(* Logix 5000 project; controller WWTP_SOLIDS_CLX vendor 1 type 14 code 54 rev 17.2; software revision 17.00; part 10 of 16 *)
(* tags used below, declared in another part *)
   Inp_PermOK : BOOL;   // 1=Permissives OK, motor can start
   Inp_NBPermOK : BOOL;   // 1=Non-Bypassable Permissives OK, motor can start
   Inp_IntlkOK : BOOL;   // 1=Interlocks OK, motor can start/run
   Inp_NBIntlkOK : BOOL;   // 1=Non-Bypassable Interlocks OK, motor can start/run
   Inp_IOFault : BOOL;   // Input Communication Status 0=OK, 1=fail
   Inp_Sim : BOOL;   // 1=Simulate working motor; 0=Start/Stop/ Monitor actual motor
   Cfg_UseRunFdbk : BOOL;   // 1=Motor run feedback should be used for failure checking
   Cfg_PCmdClear : BOOL;   // 1=Clear Program Commands on receipt 0=Leave Set
   Cfg_HasIntlkTripAlm : BOOL;   // 1=Interlock Trip Alarm exists and will be checked
   Cfg_HasIOFaultAlm : BOOL;   // 1=I/O Fault Alarm exists and will be checked
   PSet_Owner : DINT;   // Program Owner Request ID (non-zero) or Release (zero)
   PCmd_Start : BOOL;   // Program Command to Start Motor
   PCmd_Stop : BOOL;   // Program Command to Stop Motor
   PCmd_Acq : BOOL;   // Program Command to Acquire ownership (Oper/OOS to Prog)
   PCmd_Rel : BOOL;   // Program Command to Release ownership (Prog to OOS)
   PCmd_Lock : BOOL;   // Program Command to Lock Mode in Prog
   PCmd_Unlock : BOOL;   // Program Command to Unlock Mode
   PCmd_FailToStartInhibit : BOOL;   // Program Command to Inhibit Fail to Start Alarm
   PCmd_FailToStartUninhibit : BOOL;   // Program Command to Uninhibit Fail to Start Alarm
   PCmd_FailToStopInhibit : BOOL;   // Program Command to Inhibit Fail to Stop Alarm
   PCmd_FailToStopUninhibit : BOOL;   // Program Command to Uninhibit Fail to Stop Alarm
   PCmd_IntlkTripInhibit : BOOL;   // Program Command to Inhibit Interlock Trip Alarm
   PCmd_IntlkTripUninhibit : BOOL;   // Program Command to Uninhibit Interlock Trip Alarm
   PCmd_IOFaultInhibit : BOOL;   // Program Command to Inhibit I/O Fault Alarm
   PCmd_IOFaultUninhibit : BOOL;   // Program Command to Uninhibit I/O Fault Alarm
   OCmd_Start : BOOL;   // Operator Command to Start Motor
   OCmd_Stop : BOOL;   // Operator Command to Stop Motor
   OCmd_Bypass : BOOL;   // Operator Command to Bypass all Bypassable Interlocks and Permissives
   OCmd_Check : BOOL;   // Operator Command to Check (not bypass) all Interlocks and Permissives
   MCmd_Disable : BOOL;   // Maintenance Command to Disable Motor
   MCmd_Enable : BOOL;   // Maintenance Command to Enable (allow to run) Motor
   Val_Owner : DINT;   // Current Object Owner ID (0=not owned)
   Val_Notify : SINT;   // Current Alarm Level and Acknowledgement (enumeration)
   Sts_Stopped : BOOL;   // 1=Motor requested to stop and is confirmed stopped
   Sts_Starting : BOOL;   // 1=Motor requested to run and awaiting run feedback
   Sts_Running : BOOL;   // 1=Motor requested to run and is confirmed running
   Sts_Stopping : BOOL;   // 1=Motor requested to stop and awaiting stopped feedback
   Sts_Available : BOOL;   // 1=Motor available for control by automation (Prog)
   Sts_Bypass : BOOL;   // 1=Bypassable Interlocks and Permissives are Bypassed
   Sts_BypActive : BOOL;   // 1=Bypassing Active (Bypassed or Maintenance)
   Sts_Disabled : BOOL;   // 1=Motor is Disabled
   Sts_Hand : BOOL;   // 1=Mode is Hand (supersedes Maint, Ovrd, Prog, Oper)
   Sts_Maint : BOOL;   // 1=Mode is Maintenance (supersedes Ovrd, Prog, Oper)
   Sts_Prog : BOOL;   // 1=Mode is Program (auto)
   Sts_Oper : BOOL;   // 1=Mode is Operator (manual)
   Sts_FailToStop : BOOL;   // 1=Motor Failed to Stop
   Alm_IntlkTrip : BOOL;   // 1=Alarm: Motor stopped by an Interlock NOT OK
   Ack_IntlkTrip : BOOL;   // 1=Interlock Trip Alarm has been acknowledged
   Sts_IntlkTripDisabled : BOOL;   // 1=Interlock Trip Alarm is Disabled (not saved or sent)
   Sts_IntlkTripInhibited : BOOL;   // 1=Interlock Trip Alarm has been inhibited by logic
   Sts_IntlkTripSuppressed : BOOL;   // 1=Interlock Trip Alarm has been suppressed (logged only)
   Alm_IOFault : BOOL;   // 1=I/O Fault Alarm
   Ack_IOFault : BOOL;   // 1=I/O Fault Alarm has been acknowledged
   Sts_IOFaultDisabled : BOOL;   // 1=I/O Fault Alarm is Disabled (not saved or sent)
   Sts_IOFaultInhibited : BOOL;   // 1=I/O Fault Alarm has been inhibited by logic
   Sts_IOFaultSuppressed : BOOL;   // 1=I/O Fault Alarm has been suppressed (logged only)
   Rdy_Start : BOOL;   // 1=Ready to receive OCmd_Start (enables HMI button)
   Rdy_Stop : BOOL;   // 1=Ready to receive OCmd_Stop (enables HMI button)
   Rdy_Bypass : BOOL;   // 1=Ready to receive OCmd_Bypass (enables HMI button)
   Rdy_Check : BOOL;   // 1=Ready to receive OCmd_Check (enables HMI button)
   Rdy_Disable : BOOL;   // 1=Ready to receive MCmd_Disable (enables HMI button)
   Rdy_Enable : BOOL;   // 1=Ready to receive MCmd_Enable (enables HMI button)
   Mode : P_Mode;   // Motor Mode Selection
   IOFault : P_Alarm;   // I/O Fault Alarm
   IntlkTrip : P_Alarm;   // Interlock Trip Alarm
   FailToStop : P_Alarm;   // Motor Failed to Stop Alarm
   FailToStart : P_Alarm;   // Motor Failed to Start Alarm
   Wrk_Run : BOOL;   // 1=Motor should be "running", 0=should be "stopped"
   Wrk_Fault : BOOL;   // 1=a Motor Fault has been detected
   Wrk_RunFdbk : BOOL;   // Run Feedback based on mode, simulation, etc. 1=running
   Wrk_Notify : DINT;   // Buffer for building Val_Notify
   Wrk_Disabled : BOOL;   // Internal Motor is Disabled
(* P_Motor, continued *)

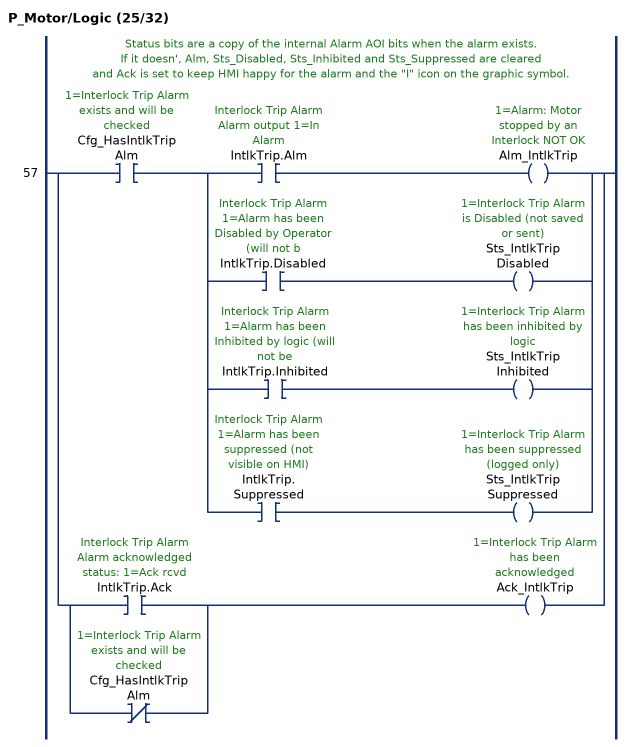
   // Status bits are a copy of the internal Alarm AOI bits when the alarm exists.
   // If it doesn', Alm, Sts_Disabled, Sts_Inhibited and Sts_Suppressed are cleared
   // and Ack is set to keep HMI happy for the alarm and the "I" icon on the graphic symbol.
   57: [XIC(Cfg_HasIntlkTripAlm) [XIC(IntlkTrip.Alm) OTE(Alm_IntlkTrip) ,XIC(IntlkTrip.Disabled) OTE(Sts_IntlkTripDisabled) ,XIC(IntlkTrip.Inhibited) OTE(Sts_IntlkTripInhibited) ,XIC(IntlkTrip.Suppressed) OTE(Sts_IntlkTripSuppressed) ] ,[XIC(IntlkTrip.Ack) ,XIO(Cfg_HasIntlkTripAlm) ] OTE(Ack_IntlkTrip) ];
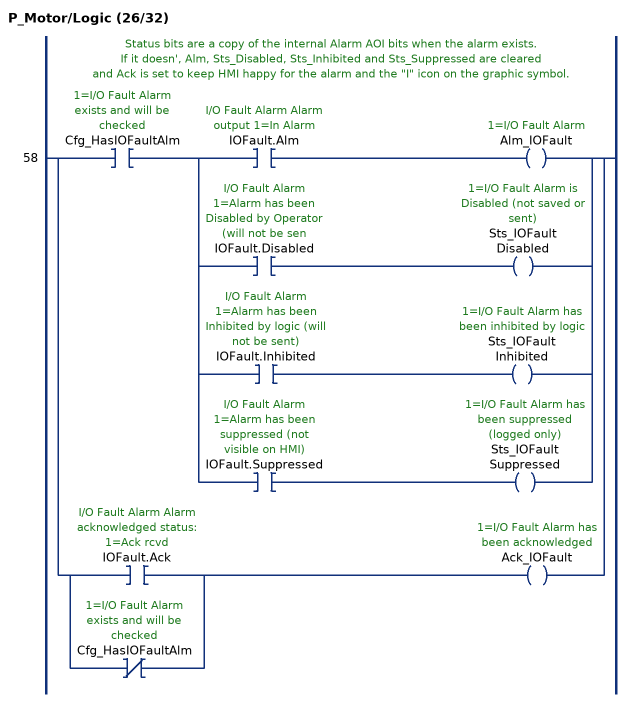
   // Status bits are a copy of the internal Alarm AOI bits when the alarm exists.
   // If it doesn', Alm, Sts_Disabled, Sts_Inhibited and Sts_Suppressed are cleared
   // and Ack is set to keep HMI happy for the alarm and the "I" icon on the graphic symbol.
   58: [XIC(Cfg_HasIOFaultAlm) [XIC(IOFault.Alm) OTE(Alm_IOFault) ,XIC(IOFault.Disabled) OTE(Sts_IOFaultDisabled) ,XIC(IOFault.Inhibited) OTE(Sts_IOFaultInhibited) ,XIC(IOFault.Suppressed) OTE(Sts_IOFaultSuppressed) ] ,[XIC(IOFault.Ack) ,XIO(Cfg_HasIOFaultAlm) ] OTE(Ack_IOFault) ];
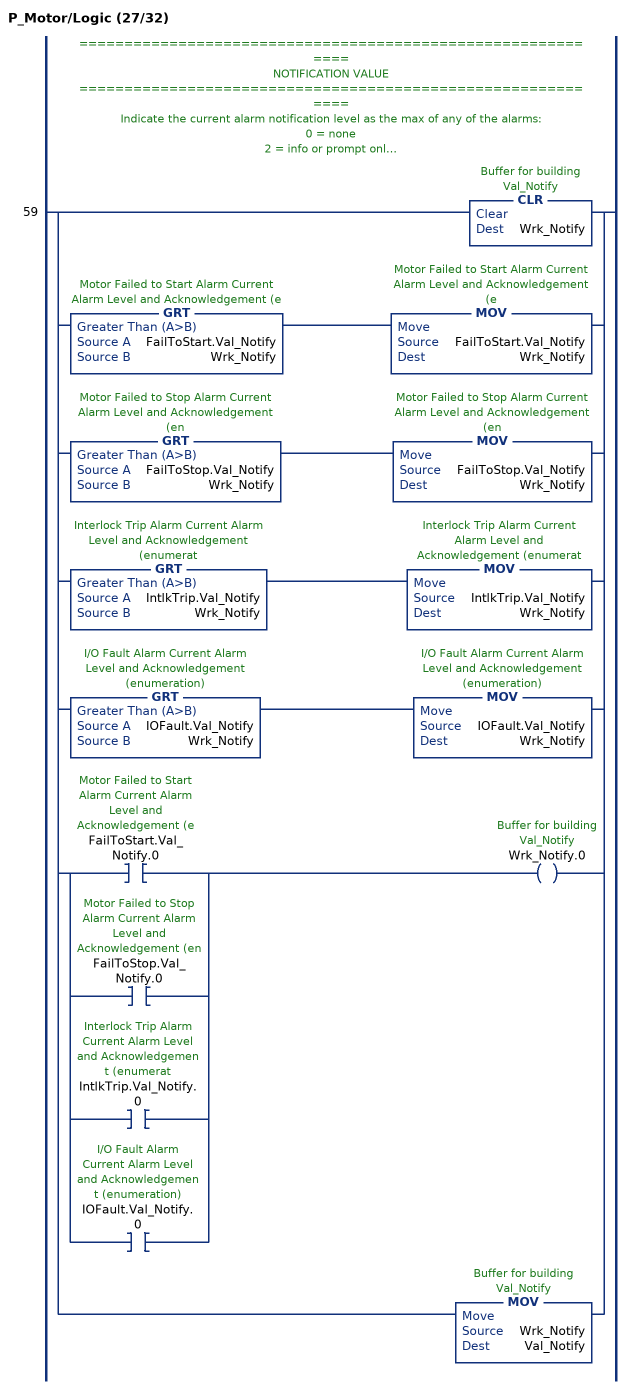
   // ============================================================
   // NOTIFICATION VALUE
   // ============================================================
   // Indicate the current alarm notification level as the max of any of the alarms:
   // 0 = none
   // 2 = info or prompt only
   // 4 = warning
   // 6 = exception (equipment impact)
   // 8 = fault (equipment failure)
   // Add one for any unsuppressed alarm that is not acknowledged (for blink).
   59: [CLR(Wrk_Notify) ,GRT(FailToStart.Val_Notify,Wrk_Notify) MOV(FailToStart.Val_Notify,Wrk_Notify) ,GRT(FailToStop.Val_Notify,Wrk_Notify) MOV(FailToStop.Val_Notify,Wrk_Notify) ,GRT(IntlkTrip.Val_Notify,Wrk_Notify) MOV(IntlkTrip.Val_Notify,Wrk_Notify) ,GRT(IOFault.Val_Notify,Wrk_Notify) MOV(IOFault.Val_Notify,Wrk_Notify) ,[XIC(FailToStart.Val_Notify.0) ,XIC(FailToStop.Val_Notify.0) ,XIC(IntlkTrip.Val_Notify.0) ,XIC(IOFault.Val_Notify.0) ] OTE(Wrk_Notify.0) ,MOV(Wrk_Notify,Val_Notify) ];
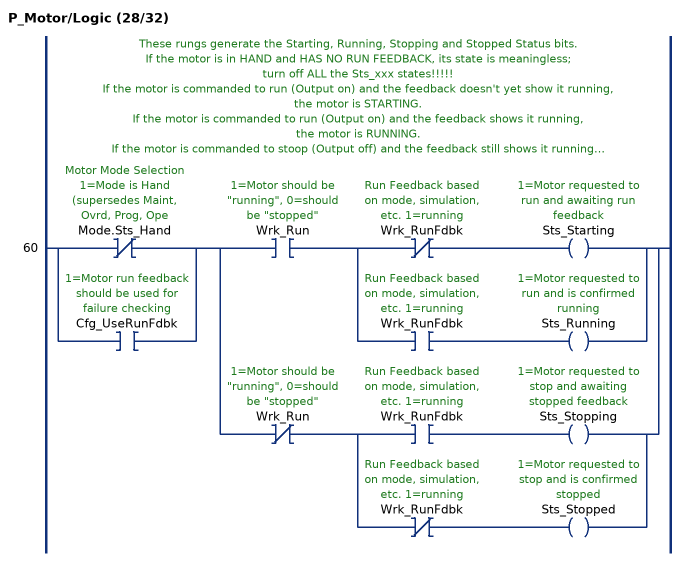
   // These rungs generate the Starting, Running, Stopping and Stopped Status bits.
   // If the motor is in HAND and HAS NO RUN FEEDBACK, its state is meaningless;
   // turn off ALL the Sts_xxx states!!!!!
   // If the motor is commanded to run (Output on) and the feedback doesn't yet show it running,
   // the motor is STARTING.
   // If the motor is commanded to run (Output on) and the feedback shows it running,
   // the motor is RUNNING.
   // If the motor is commanded to stoop (Output off) and the feedback still shows it running,
   // the motor is STOPPING.
   // If the motor is commanded to stop (Output off) and the feedback shows it has stopped,
   // the motor is STOPPED.
   60: [XIO(Mode.Sts_Hand) ,XIC(Cfg_UseRunFdbk) ][XIC(Wrk_Run) [XIO(Wrk_RunFdbk) OTE(Sts_Starting) ,XIC(Wrk_RunFdbk) OTE(Sts_Running) ] ,XIO(Wrk_Run) [XIC(Wrk_RunFdbk) OTE(Sts_Stopping) ,XIO(Wrk_RunFdbk) OTE(Sts_Stopped) ] ];
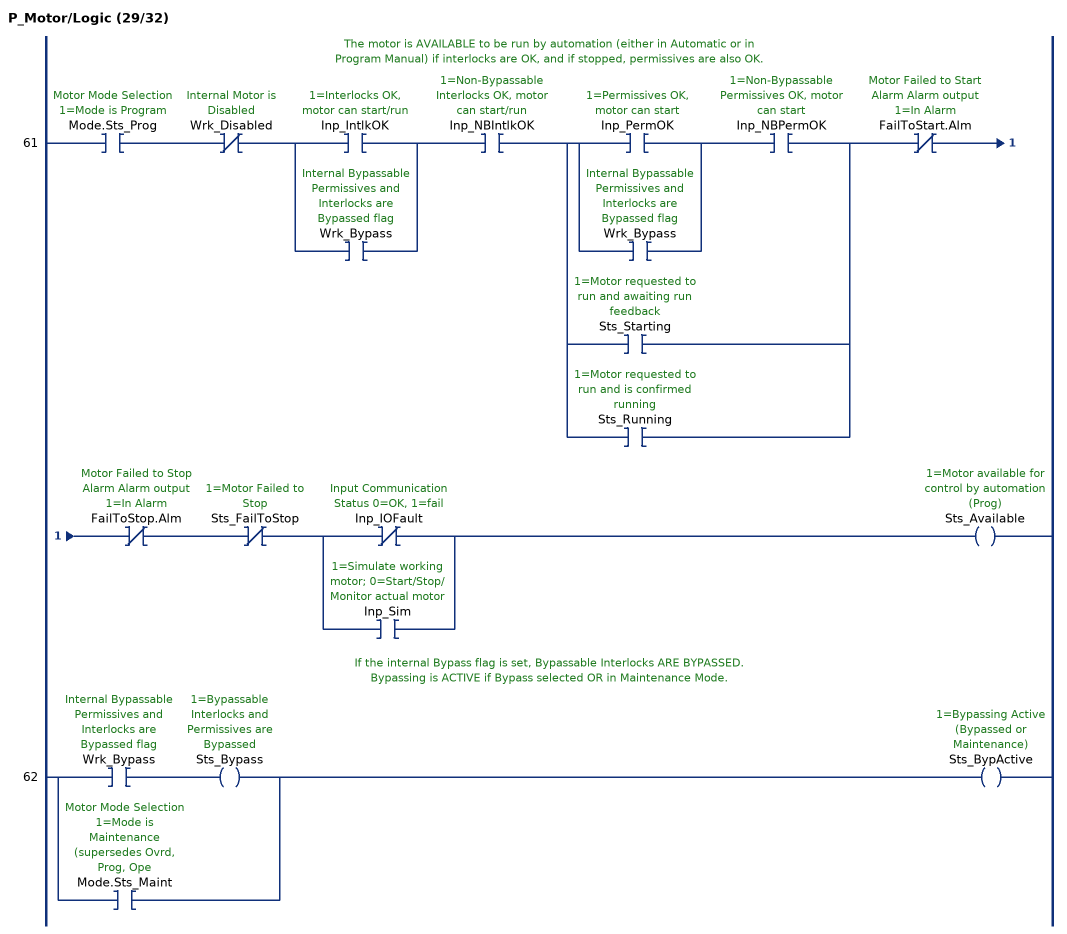
   // The motor is AVAILABLE to be run by automation (either in Automatic or in
   // Program Manual) if interlocks are OK, and if stopped, permissives are also OK.
   61: XIC(Mode.Sts_Prog)XIO(Wrk_Disabled)[XIC(Inp_IntlkOK) ,XIC(Wrk_Bypass) ]XIC(Inp_NBIntlkOK)[[XIC(Inp_PermOK) ,XIC(Wrk_Bypass) ] XIC(Inp_NBPermOK) ,XIC(Sts_Starting) ,XIC(Sts_Running) ]XIO(FailToStart.Alm)XIO(FailToStop.Alm)XIO(Sts_FailToStop)[XIO(Inp_IOFault) ,XIC(Inp_Sim) ]OTE(Sts_Available);
   // If the internal Bypass flag is set, Bypassable Interlocks ARE BYPASSED.
   // Bypassing is ACTIVE if Bypass selected OR in Maintenance Mode.
   62: [XIC(Wrk_Bypass) OTE(Sts_Bypass) ,XIC(Mode.Sts_Maint) ]OTE(Sts_BypActive);
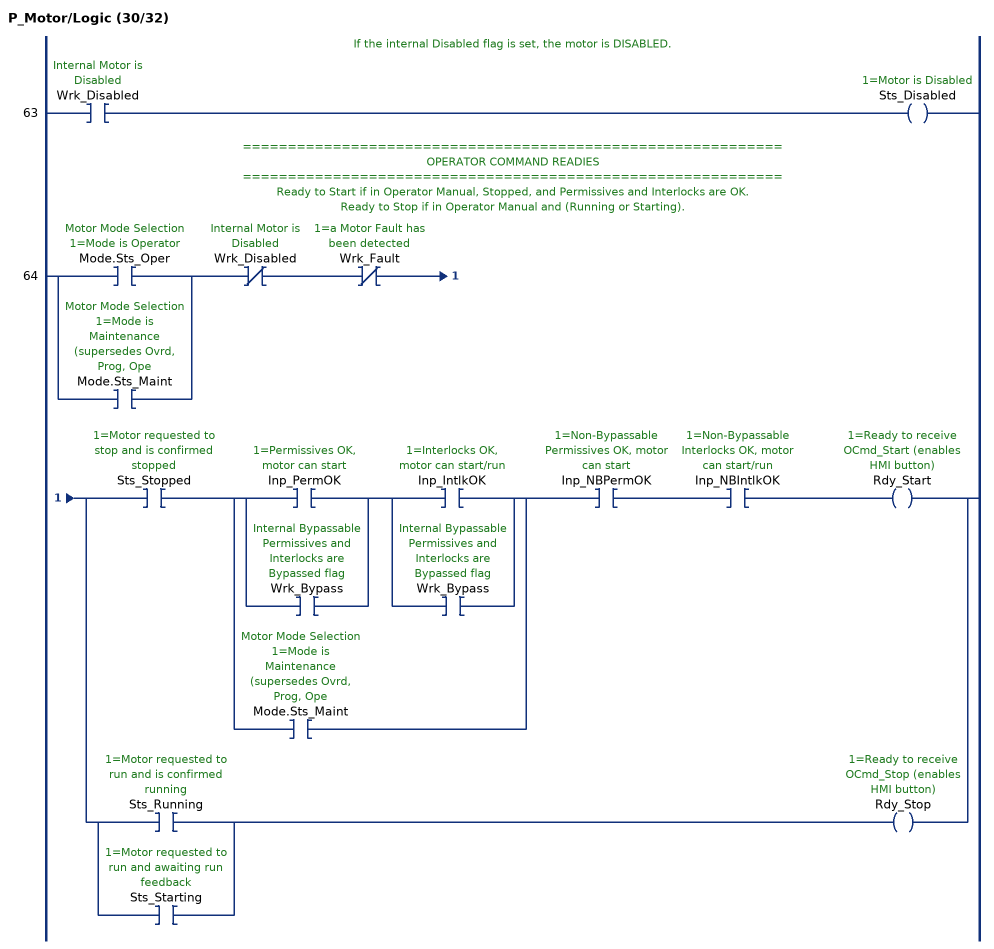
   // If the internal Disabled flag is set, the motor is DISABLED.
   63: XIC(Wrk_Disabled)OTE(Sts_Disabled);
   // ============================================================
   // OPERATOR COMMAND READIES
   // ============================================================
   // Ready to Start if in Operator Manual, Stopped, and Permissives and Interlocks are OK.
   // Ready to Stop if in Operator Manual and (Running or Starting).
   64: [XIC(Mode.Sts_Oper) ,XIC(Mode.Sts_Maint) ]XIO(Wrk_Disabled)XIO(Wrk_Fault)[XIC(Sts_Stopped) [[XIC(Inp_PermOK) ,XIC(Wrk_Bypass) ] [XIC(Inp_IntlkOK) ,XIC(Wrk_Bypass) ] ,XIC(Mode.Sts_Maint) ] XIC(Inp_NBPermOK) XIC(Inp_NBIntlkOK) OTE(Rdy_Start) ,[XIC(Sts_Running) ,XIC(Sts_Starting) ] OTE(Rdy_Stop) ];
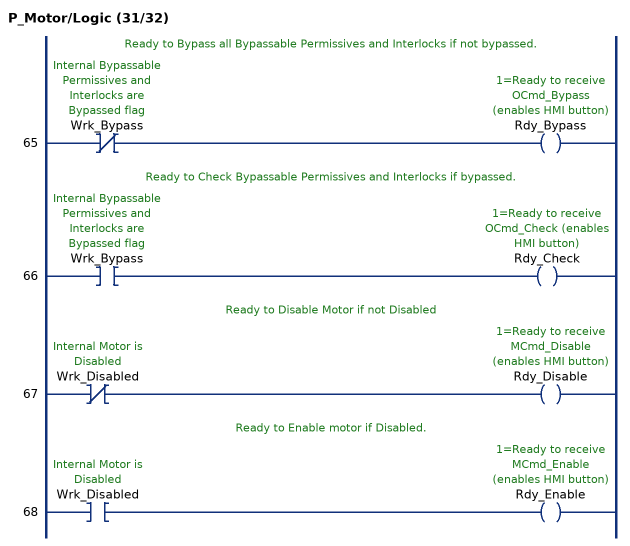
   // Ready to Bypass all Bypassable Permissives and Interlocks if not bypassed.
   65: XIO(Wrk_Bypass)OTE(Rdy_Bypass);
   // Ready to Check Bypassable Permissives and Interlocks if bypassed.
   66: XIC(Wrk_Bypass)OTE(Rdy_Check);
   // Ready to Disable Motor if not Disabled
   67: XIO(Wrk_Disabled)OTE(Rdy_Disable);
   // Ready to Enable motor if Disabled.
   68: XIC(Wrk_Disabled)OTE(Rdy_Enable);
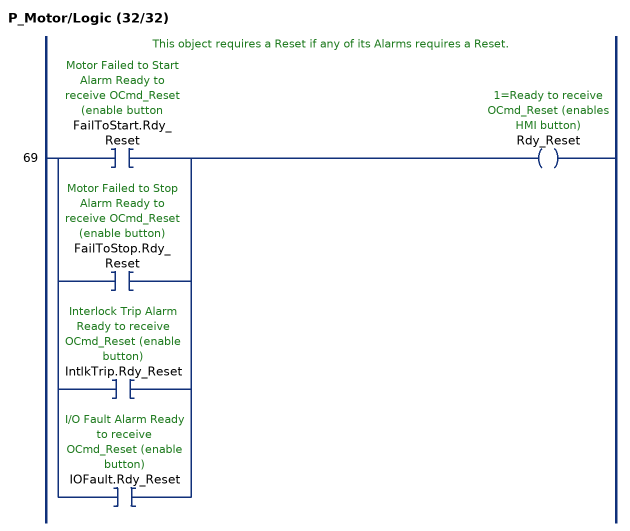
   // This object requires a Reset if any of its Alarms requires a Reset.
   69: [XIC(FailToStart.Rdy_Reset) ,XIC(FailToStop.Rdy_Reset) ,XIC(IntlkTrip.Rdy_Reset) ,XIC(IOFault.Rdy_Reset) ]OTE(Rdy_Reset);
END_ROUTINE

ROUTINE Prescan   (* ladder *)
// Clear Ownership, clear "lurking" Commands
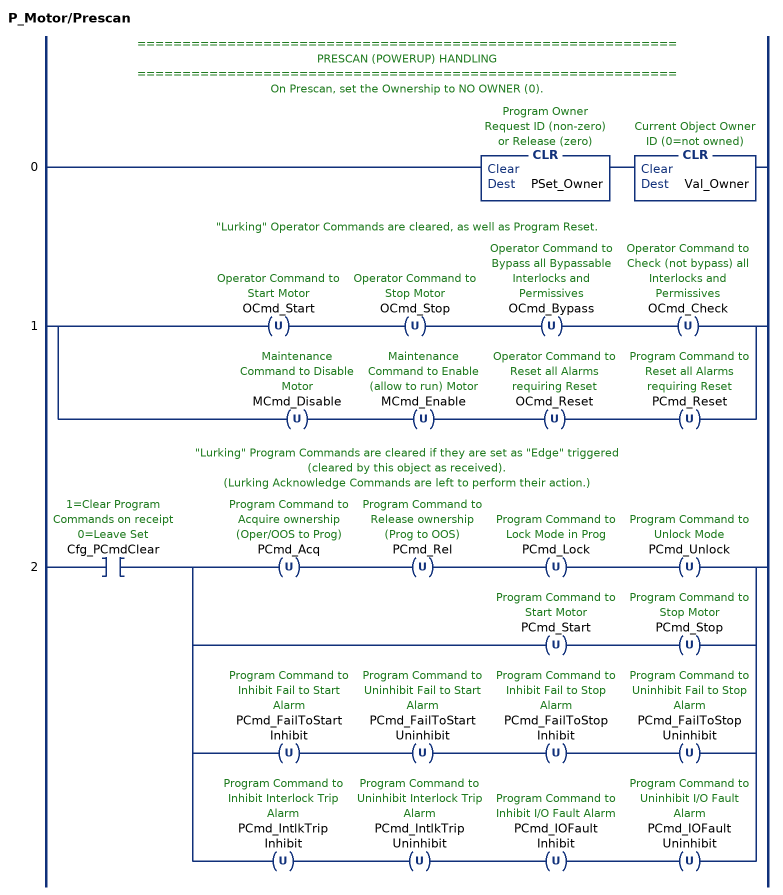
   // ============================================================
   // PRESCAN (POWERUP) HANDLING
   // ============================================================
   // On Prescan, set the Ownership to NO OWNER (0).
   0: CLR(PSet_Owner)CLR(Val_Owner);
   // "Lurking" Operator Commands are cleared, as well as Program Reset.
   1: [OTU(OCmd_Start) OTU(OCmd_Stop) OTU(OCmd_Bypass) OTU(OCmd_Check) ,OTU(MCmd_Disable) OTU(MCmd_Enable) OTU(OCmd_Reset) OTU(PCmd_Reset) ];
   // "Lurking" Program Commands are cleared if they are set as "Edge" triggered
   // (cleared by this object as received).
   // (Lurking Acknowledge Commands are left to perform their action.)
   2: XIC(Cfg_PCmdClear)[OTU(PCmd_Acq) OTU(PCmd_Rel) OTU(PCmd_Lock) OTU(PCmd_Unlock) ,OTU(PCmd_Start) OTU(PCmd_Stop) ,OTU(PCmd_FailToStartInhibit) OTU(PCmd_FailToStartUninhibit) OTU(PCmd_FailToStopInhibit) OTU(PCmd_FailToStopUninhibit) ,OTU(PCmd_IntlkTripInhibit) OTU(PCmd_IntlkTripUninhibit) OTU(PCmd_IOFaultInhibit) OTU(PCmd_IOFaultUninhibit) ];
END_ROUTINE
END_ADD_ON_INSTRUCTION

ADD_ON_INSTRUCTION P_Perm   (* revision 0.8, ExecuteEnableInFalse *)
// Permissives
// Revision note:
// Aligned name, description and local STRING values, sizes, across instructions.
// Help:
// This Instruction monitors up to 16 Permissive conditions.  It provides these features:
// *  Permissives may be configured as Bypassable.  Separate Permissives OK and
//     Non-Bypassable Permissives OK status bits are provided.
// Only Permissives configured as Bypassable should be bypassed.  This is determined
// by the object using this instruction's status bits.  Bypassable Permissives might be
// bypassed in Maintenance Mode or by command from a Maintenance faceplate.
VAR_INPUT
   Inp_Perm00 : BOOL := 1; {visible}   // Permissive Cond 00 (1=OK,0=don't start)
   Inp_Perm01 : BOOL := 1; {visible}   // Permissive Cond 01 (1=OK,0=don't start)
   Inp_Perm02 : BOOL := 1; {visible}   // Permissive Cond 02 (1=OK,0=don't start)
   Inp_Perm03 : BOOL := 1; {visible}   // Permissive Cond 03 (1=OK,0=don't start)
   Inp_Perm04 : BOOL := 1; {visible}   // Permissive Cond 04 (1=OK,0=don't start)
   Inp_Perm05 : BOOL := 1; {visible}   // Permissive Cond 05 (1=OK,0=don't start)
   Inp_Perm06 : BOOL := 1; {visible}   // Permissive Cond 06 (1=OK,0=don't start)
   Inp_Perm07 : BOOL := 1; {visible}   // Permissive Cond 07 (1=OK,0=don't start)
   Inp_Perm08 : BOOL := 1;   // Permissive Cond 08 (1=OK,0=don't start)
   Inp_Perm09 : BOOL := 1;   // Permissive Cond 09 (1=OK,0=don't start)
   Inp_Perm10 : BOOL := 1;   // Permissive Cond 10 (1=OK,0=don't start)
   Inp_Perm11 : BOOL := 1;   // Permissive Cond 11 (1=OK,0=don't start)
   Inp_Perm12 : BOOL := 1;   // Permissive Cond 12 (1=OK,0=don't start)
   Inp_Perm13 : BOOL := 1;   // Permissive Cond 13 (1=OK,0=don't start)
   Inp_Perm14 : BOOL := 1;   // Permissive Cond 14 (1=OK,0=don't start)
   Inp_Perm15 : BOOL := 1;   // Permissive Cond 15 (1=OK,0=don't start)
   Cfg_Bypassable : INT;   // Set bits indicate which conditions can be bypassed
END_VAR
VAR_OUTPUT
   Sts_PermOK : BOOL := 1; {visible}   // Overall Permissive Status (1=OK to start)
   Sts_NBPermOK : BOOL := 1; {visible}   // Non-Bypassable Permissive Status (1 =all non- bypassable Permissives OK to start)
   Sts_Perm : INT := 2#1111_1111_1111_1111; {visible}   // Individual Permissive Status (1=OK, 0=don't start)
END_VAR
VAR
   Cfg_CondTxt : STRING_20[16] := ([0] := 'Permissive 0');   // Short HMI description of Permissive Conditions
   Wrk_Inp : INT;   // Collection copy of Inp_PermXXs
   Wrk_Bypass : INT;   // Working Register for Bypassable Permissives
END_VAR

ROUTINE EnableInFalse   (* ladder *)
// Set summary "OK" Status bits to FALSE (0)
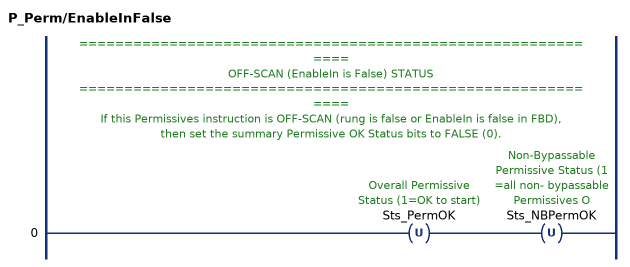
   // ============================================================
   // OFF-SCAN (EnableIn is False) STATUS
   // ============================================================
   // If this Permissives instruction is OFF-SCAN (rung is false or EnableIn is false in FBD),
   // then set the summary Permissive OK Status bits to FALSE (0).
   0: OTU(Sts_PermOK)OTU(Sts_NBPermOK);
END_ROUTINE

ROUTINE Logic   (* ladder *)
// Check Permissive Conditions
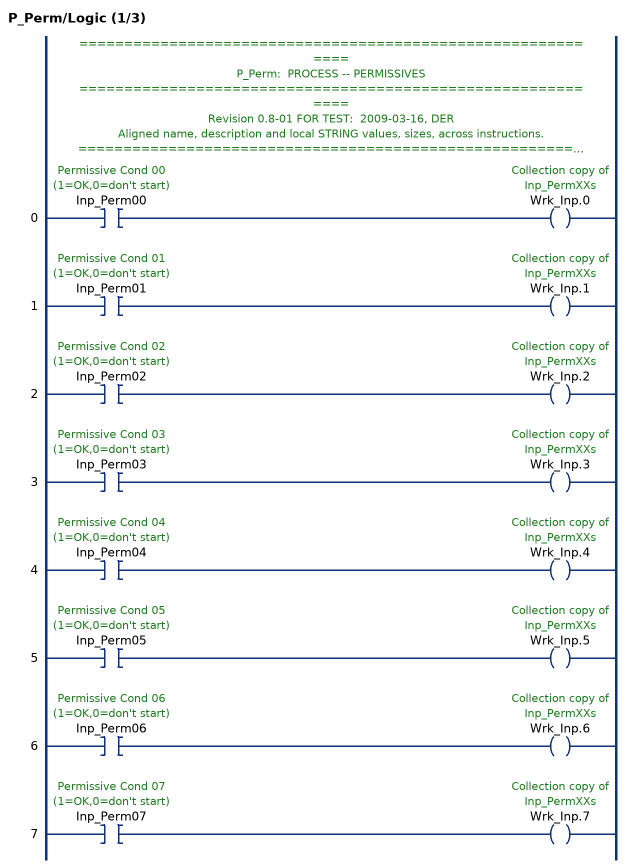
   // ============================================================
   // P_Perm:  PROCESS -- PERMISSIVES
   // ============================================================
   // Revision 0.8-01 FOR TEST:  2009-03-16, DER
   // Aligned name, description and local STRING values, sizes, across instructions.
   // ============================================================
   // This Instruction monitors up to 16 Permissive conditions.  It provides these features:
   // *  Permissives may be configured as Bypassable.  A separate Sts_NBPermOK
   // (Non-Bypassable Permissives OK) status is provided, which the destination
   // object can use forBypass, Maintenance and other functions,
   // where Bypassable Permissives can be ignored.
   // ============================================================
   // POWERUP / INVALID STATE HANDLING
   // ============================================================
   // No special powerup code is required for this object.
   // ============================================================
   // INPUT GATHERING
   // ============================================================
   // This object uses word-wise logic.  The first 16 rungs collect the individual
   // Permissive Inputs together into a 16-bit integer word for word-wise processing.
   0: XIC(Inp_Perm00)OTE(Wrk_Inp.0);
   1: XIC(Inp_Perm01)OTE(Wrk_Inp.1);
   2: XIC(Inp_Perm02)OTE(Wrk_Inp.2);
   3: XIC(Inp_Perm03)OTE(Wrk_Inp.3);
   4: XIC(Inp_Perm04)OTE(Wrk_Inp.4);
   5: XIC(Inp_Perm05)OTE(Wrk_Inp.5);
   6: XIC(Inp_Perm06)OTE(Wrk_Inp.6);
   7: XIC(Inp_Perm07)OTE(Wrk_Inp.7);
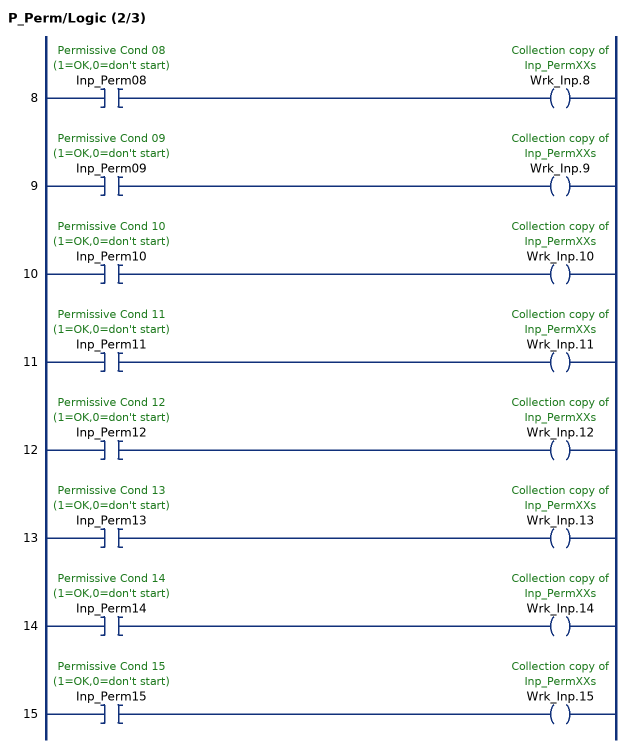
   8: XIC(Inp_Perm08)OTE(Wrk_Inp.8);
   9: XIC(Inp_Perm09)OTE(Wrk_Inp.9);
   10: XIC(Inp_Perm10)OTE(Wrk_Inp.10);
   11: XIC(Inp_Perm11)OTE(Wrk_Inp.11);
   12: XIC(Inp_Perm12)OTE(Wrk_Inp.12);
   13: XIC(Inp_Perm13)OTE(Wrk_Inp.13);
   14: XIC(Inp_Perm14)OTE(Wrk_Inp.14);
   15: XIC(Inp_Perm15)OTE(Wrk_Inp.15);
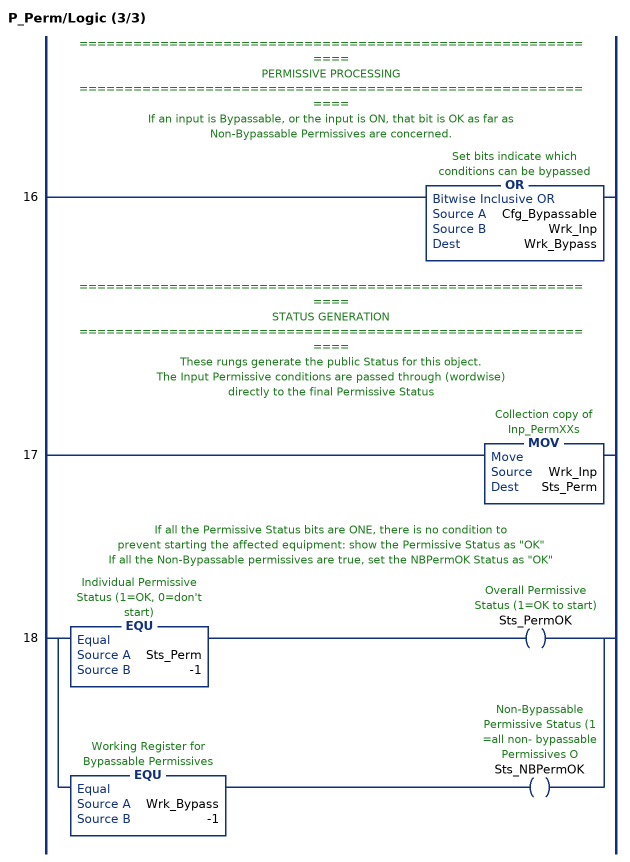
   // ============================================================
   // PERMISSIVE PROCESSING
   // ============================================================
   // If an input is Bypassable, or the input is ON, that bit is OK as far as
   // Non-Bypassable Permissives are concerned.
   16: OR(Cfg_Bypassable,Wrk_Inp,Wrk_Bypass);
   // ============================================================
   // STATUS GENERATION
   // ============================================================
   // These rungs generate the public Status for this object.
   // The Input Permissive conditions are passed through (wordwise)
   // directly to the final Permissive Status
   17: MOV(Wrk_Inp,Sts_Perm);
   // If all the Permissive Status bits are ONE, there is no condition to
   // prevent starting the affected equipment: show the Permissive Status as "OK"
   // If all the Non-Bypassable permissives are true, set the NBPermOK Status as "OK"
   18: [EQU(Sts_Perm,-1) OTE(Sts_PermOK) ,EQU(Wrk_Bypass,-1) OTE(Sts_NBPermOK) ];
END_ROUTINE
END_ADD_ON_INSTRUCTION

ADD_ON_INSTRUCTION P_Reset   (* revision 0.6, ExecutePrescan, ExecuteEnableInFalse *)
// Reset
// Revision note:
// Aligned name, description and local STRING values, sizes, across instructions.
// Help:
// This instruction provides a central point in a control strategy (CM, EM, Unit, Group, Cell, Area, etc.)
// or controller for accepting and fanning out a Reset of equipment alarms and faults.
// Resets are accepted from Program Command (PCmd_Reset), Operator Command (OCmd_Reset) or
// as an Input from another object (Inp_Reset).  The input can be tied to the output of a higher-level
// Reset instruction to cascade Resets down through a hierarchy, say from a master Station Reset
// to individual groups or units.
// The minimum duration of the reset Output is configurable.  This can be set to allow time for a
// Reset sent to equipment via an output card to feed back into the system via inputs.
// The P_Reset instruction can be used on a ladder rung with the rung condition transitioning
// from FALSE to TRUE causing the output to pulse.  In this configuration, the Program and
// Operator Commands and the reset Input still function normally, even if the rung is FALSE.
VAR_INPUT
   Inp_Reset : BOOL; {visible}   // Reset Input, 1=Reset, from pushbutton or another object
   Inp_ResetReqd : BOOL := 1; {visible}   // 1=Reset Required, enable Reset button
   Cfg_MinHoldTime : DINT := 1;   // Minimum Time to hold Reset Output true (sec)
   PCmd_Reset : BOOL;   // Program Command to Reset, from other object
   OCmd_Reset : BOOL;   // Operator Command to Reset, from HMI
END_VAR
VAR_OUTPUT
   Out_Reset : BOOL; {visible}   // 1=Reset received for this P_Reset's scope
   Sts_Err : BOOL; {visible}   // 1=Error in Config: Invalid Hold Time (use 0 to 2147483)
   Rdy_Reset : BOOL := 1;   // 1=Ready to receive OCmd_Reset (enable button)
END_VAR
VAR
   Wrk_HoldT : TIMER;   // Reset Output Hold Timer (TOF)
   Wrk_EnableInONS : BOOL := 1;   // EnableIn transition detection to pulse Reset Output
   Wrk_HoldONS : BOOL;   // One-Shot to fire Hold Timer to ensure min. output ON time.
   Wrk_ResetCond : BOOL;   // Any incoming Reset condition is TRUE
END_VAR

ROUTINE EnableInFalse   (* ladder *)
// Sets up for One-Shot trigger of Reset using XIC/XIO on rung
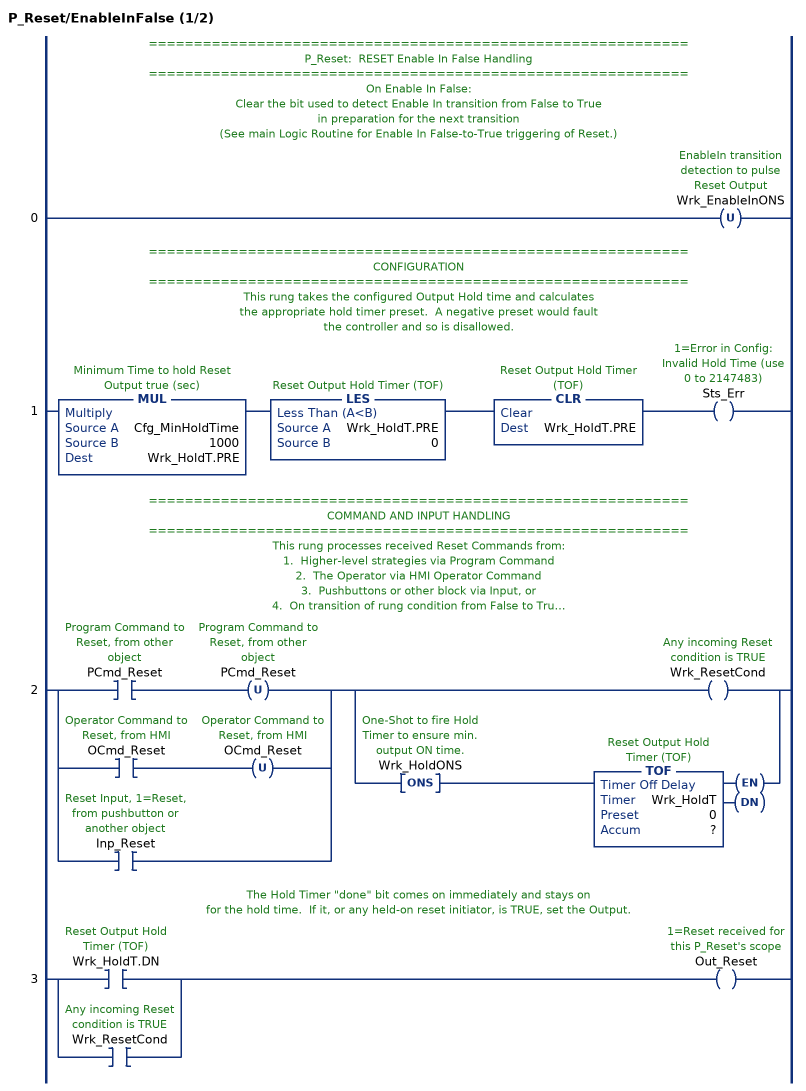
   // ============================================================
   // P_Reset:  RESET Enable In False Handling
   // ============================================================
   // On Enable In False:
   // Clear the bit used to detect Enable In transition from False to True
   // in preparation for the next transition
   // (See main Logic Routine for Enable In False-to-True triggering of Reset.)
   0: OTU(Wrk_EnableInONS);
   // ============================================================
   // CONFIGURATION
   // ============================================================
   // This rung takes the configured Output Hold time and calculates
   // the appropriate hold timer preset.  A negative preset would fault
   // the controller and so is disallowed.
   1: MUL(Cfg_MinHoldTime,1000,Wrk_HoldT.PRE)LES(Wrk_HoldT.PRE,0)CLR(Wrk_HoldT.PRE)OTE(Sts_Err);
   // ============================================================
   // COMMAND AND INPUT HANDLING
   // ============================================================
   // This rung processes received Reset Commands from:
   // 1.  Higher-level strategies via Program Command
   // 2.  The Operator via HMI Operator Command
   // 3.  Pushbuttons or other block via Input, or
   // 4.  On transition of rung condition from False to True
   // (button or other logic as rung condition).
   // The reset starts the Hold Timer (One-Shot Off-Delay)
   // to ensure the output is held on for at least the minimum time.
   2: [XIC(PCmd_Reset) OTU(PCmd_Reset) ,XIC(OCmd_Reset) OTU(OCmd_Reset) ,XIC(Inp_Reset) ][OTE(Wrk_ResetCond) ,ONS(Wrk_HoldONS) TOF(Wrk_HoldT,?,?) ];
   // The Hold Timer "done" bit comes on immediately and stays on
   // for the hold time.  If it, or any held-on reset initiator, is TRUE, set the Output.
   3: [XIC(Wrk_HoldT.DN) ,XIC(Wrk_ResetCond) ]OTE(Out_Reset);
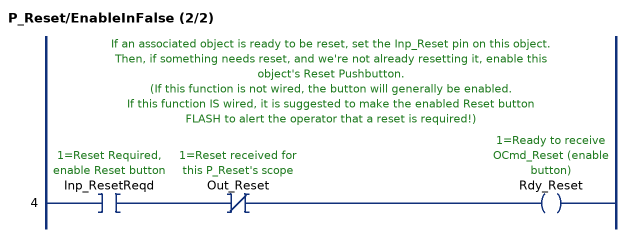
   // If an associated object is ready to be reset, set the Inp_Reset pin on this object.
   // Then, if something needs reset, and we're not already resetting it, enable this
   // object's Reset Pushbutton.
   // (If this function is not wired, the button will generally be enabled.
   // If this function IS wired, it is suggested to make the enabled Reset button
   // FLASH to alert the operator that a reset is required!)
   4: XIC(Inp_ResetReqd)XIO(Out_Reset)OTE(Rdy_Reset);
END_ROUTINE

ROUTINE Logic   (* ladder *)
// Process Reset Input and Commands
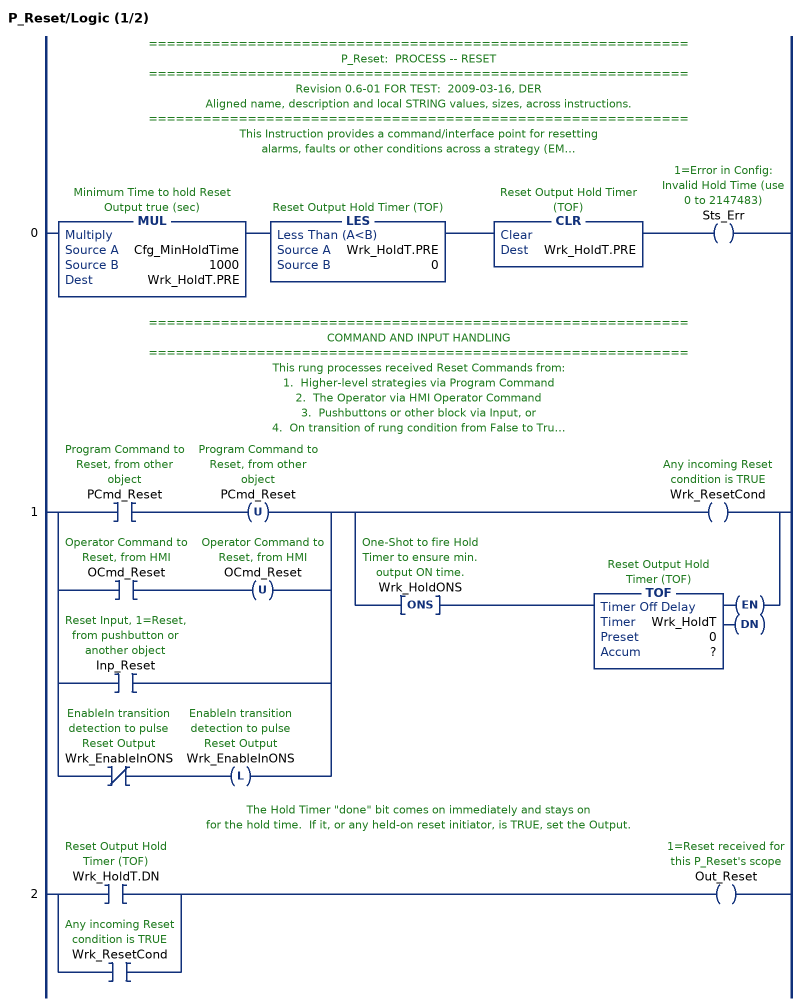
   // ============================================================
   // P_Reset:  PROCESS -- RESET
   // ============================================================
   // Revision 0.6-01 FOR TEST:  2009-03-16, DER
   // Aligned name, description and local STRING values, sizes, across instructions.
   // ============================================================
   // This Instruction provides a command/interface point for resetting
   // alarms, faults or other conditions across a strategy (EM,
   // Unit, Cell, Area, Site, etc.).  Its Output is intended to be wired
   // to input, device and interlock instructions to allow a single reset
   // command or pushbutton to reset alarms and faults in all objects in its scope.
   // ============================================================
   // POWER UP OR INVALID STATE
   // ============================================================
   // No special power up logic is required.
   // ============================================================
   // CONFIGURATION
   // ============================================================
   // This rung takes the configured Output Hold time and calculates
   // the appropriate hold timer preset.  A negative preset would fault
   // the controller and so is disallowed and flagged.
   0: MUL(Cfg_MinHoldTime,1000,Wrk_HoldT.PRE)LES(Wrk_HoldT.PRE,0)CLR(Wrk_HoldT.PRE)OTE(Sts_Err);
   // ============================================================
   // COMMAND AND INPUT HANDLING
   // ============================================================
   // This rung processes received Reset Commands from:
   // 1.  Higher-level strategies via Program Command
   // 2.  The Operator via HMI Operator Command
   // 3.  Pushbuttons or other block via Input, or
   // 4.  On transition of rung condition from False to True
   // (button or other logic as rung condition).
   // The reset starts the Hold Timer (One-Shot Off-Delay)
   // to ensure the output is held on for at least the minimum time.
   1: [XIC(PCmd_Reset) OTU(PCmd_Reset) ,XIC(OCmd_Reset) OTU(OCmd_Reset) ,XIC(Inp_Reset) ,XIO(Wrk_EnableInONS) OTL(Wrk_EnableInONS) ][OTE(Wrk_ResetCond) ,ONS(Wrk_HoldONS) TOF(Wrk_HoldT,?,?) ];
   // The Hold Timer "done" bit comes on immediately and stays on
   // for the hold time.  If it, or any held-on reset initiator, is TRUE, set the Output.
   2: [XIC(Wrk_HoldT.DN) ,XIC(Wrk_ResetCond) ]OTE(Out_Reset);
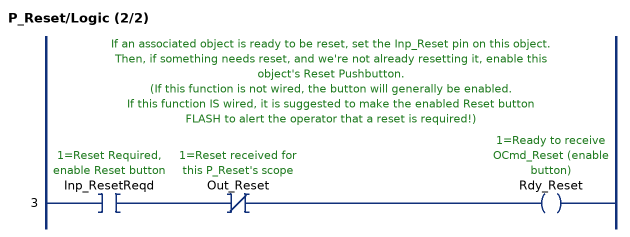
   // If an associated object is ready to be reset, set the Inp_Reset pin on this object.
   // Then, if something needs reset, and we're not already resetting it, enable this
   // object's Reset Pushbutton.
   // (If this function is not wired, the button will generally be enabled.
   // If this function IS wired, it is suggested to make the enabled Reset button
   // FLASH to alert the operator that a reset is required!)
   3: XIC(Inp_ResetReqd)XIO(Out_Reset)OTE(Rdy_Reset);
END_ROUTINE

ROUTINE Prescan   (* ladder *)
// Clear "lurking" Commands
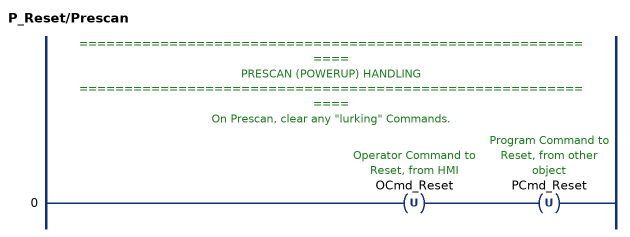
   // ============================================================
   // PRESCAN (POWERUP) HANDLING
   // ============================================================
   // On Prescan, clear any "lurking" Commands.
   0: OTU(OCmd_Reset)OTU(PCmd_Reset);
END_ROUTINE
END_ADD_ON_INSTRUCTION
